{attribute 'GeneratedUsingTerminal: AES-D-BC-ECAT Gen2-0001'}
{attribute addProperty BoxType "AES-D-BC-ECAT Gen2-0001"}
{attribute addProperty Id "digital_Data_OAT %Q*ARRAY[0..3] OF ARRAY[0..7] OF BOOL"}
{attribute addProperty CRC "2104334051"}
{attribute addProperty Size "4"}
TYPE AES_D_BC_ECAT_Gen2_4bytes_Data_Outputs EXTENDS TcoIo.OutputBase_10CEE7DE :
STRUCT
	{attribute addProperty Name "digital_Data_O"}
	digital_Data_O AT %Q* : ARRAY[0..3] OF ARRAY[0..7] OF BOOL;
END_STRUCT
END_TYPE

(* stored: Version 1.1.0.1
   DUT AES_D_BC_ECAT_Gen2_4bytes_Data_Outputs: Id {2aff5cd9-5bf3-49b8-b1ff-7a46e17e7927} *)
